{attribute addProperty BoxType "EK1100-0000-0018"}
{attribute addProperty Id "Beckhoff_EL31xxEK1122Beckhoff_EL31xxEK1122_F35612A4162A_0001_EL3101_0000_0016EL3101_EA8DF7B012816A_0002_EL3101_0000_0017EL3101_EA8DF7B012816A_0003_EL3101_0000_0018EL3101_60464DCF12816A_0004_EL3101_0000_0019EL3101_60464DCF12816A_0005_EL3102_0000_0000EL3102_B73BDD5814418A_0006_EL3102_0000_0016EL3102_8E42B51D24430.5A_0007_EL3102_0000_0017EL3102_8E42B51D24430.5A_0008_EL3102_0000_0018EL3102_8E42B51D24430.5A_0009_EL3102_0000_0019EL3102_68FCBB3024430.5A_0010_EL3102_0000_0020EL3102_1C870F0C16020A_0011_EL3104_0000_0016EL3104_55F04E9922428A_0012_EL3104_0000_0017EL3104_55F04E9922428A_0013_EL3104_0000_0018EL3104_83515A0D22428A_0014_EL3104_0000_0019EL3104_83515A0D22428A_0015_EL3104_0000_0020EL3104_83515A0D22428A_0016_EL3111_0000_0016EL3111_EA8DF7B012816A_0017_EL3111_0000_0017EL3111_EA8DF7B012816A_0018_EL3111_0000_0018EL3111_60464DCF12816A_0019_EL3111_0000_0019EL3111_60464DCF12816A_0020_EL3111_0000_0020EL3111_60464DCF12816A_0021_EL3112_0000_0000EL3112_B73BDD5814418A_0022_EL3112_0000_0016EL3112_8E42B51D24430.5A_0023_EL3112_0000_0017EL3112_8E42B51D24430.5A_0024_EL3112_0000_0018EL3112_8E42B51D24430.5A_0025_EL3112_0000_0019EL3112_1C870F0C16020A_0026_EL3112_0011_0016EL3112_1C870F0C16020A_0027_EL3114_0000_0016EL3114_129272B139249A_0028_EL3114_0000_0017EL3114_55F04E9922428A_0029_EL3114_0000_0018EL3114_55F04E9922428A_0030_EL3114_0000_0019EL3114_83515A0D22428A_0031_EL3114_0000_0020EL3114_83515A0D22428A_0032_EL3114_0000_0021EL3114_83515A0D22428A_0033_EL3121_0000_0016EL3121_EA8DF7B012816A_0034_EL3121_0000_0017EL3121_EA8DF7B012816A_0035_EL3121_0000_0018EL3121_60464DCF12816A_0036_EL3121_0000_0019EL3121_60464DCF12816A_0037_EL3122_0000_0000EL3122_B73BDD5814418A_0038_EL3122_0000_0016EL3122_8E42B51D24430.5A_0039_EL3122_0000_0017EL3122_8E42B51D24430.5A_0040_EL3122_0000_0018EL3122_8E42B51D24430.5A_0041_EL3122_0000_0019EL3122_1C870F0C16020A_0042_EL3124_0000_0016EL3124_55F04E9922428A_0043_EL3124_0000_0017EL3124_55F04E9922428A_0044_EL3124_0000_0018EL3124_83515A0D22428A_0045_EL3124_0000_0019EL3124_83515A0D22428A_0046_EL3124_0000_0020EL3124_83515A0D22428A_0047_EL3124_0090_0016EL3124_83515A0D22428A_0048_EL3141_0000_0016EL3141_EA8DF7B012816A_0049_EL3141_0000_0017EL3141_EA8DF7B012816A_0050_EL3141_0000_0018EL3141_60464DCF12816A_0051_EL3141_0000_0019EL3141_60464DCF12816A_0052_EL3141_0000_0020EL3141_60464DCF12816A_0053_EL3142_0000_0000EL3142_B73BDD5814418A_0054_EL3142_0000_0016EL3142_8E42B51D24430.5A_0055_EL3142_0000_0017EL3142_8E42B51D24430.5A_0056_EL3142_0000_0018EL3142_8E42B51D24430.5A_0057_EL3142_0000_0019EL3142_1C870F0C16020A_0058_EL3142_0010_0000EL3142_B73BDD5814418A_0059_EL3142_0010_0016EL3142_8E42B51D24430.5A_0060_EL3142_0010_0017EL3142_8E42B51D24430.5A_0061_EL3142_0010_0018EL3142_8E42B51D24430.5A_0062_EL3142_0010_0019EL3142_8E42B51D24430.5A_0063_EL3142_0010_0020EL3142_1C870F0C16020A_0064_EL3142_0010_0021EL3142_1C870F0C16020A_0065_EL3144_0000_0016EL3144_55F04E9922428A_0066_EL3144_0000_0017EL3144_55F04E9922428A_0067_EL3144_0000_0018EL3144_83515A0D22428A_0068_EL3144_0000_0019EL3144_83515A0D22428A_0069_EL3144_0000_0020EL3144_83515A0D22428A_0070_EL3151_0000_0016EL3151_50D9316A17021.25A_0071_EL3151_0000_0017EL3151_50D9316A17021.25A_0072_EL3151_0000_0018EL3151_60464DCF12816A_0073_EL3151_0000_0019EL3151_60464DCF12816A_0074_EL3151_0000_0020EL3151_60464DCF12816A_0075_EL3152_0000_0000EL3152_B73BDD5814418A_0076_EL3152_0000_0016EL3152_8E42B51D24430.5A_0077_EL3152_0000_0017EL3152_8E42B51D24430.5A_0078_EL3152_0000_0018EL3152_8E42B51D24430.5A_0079_EL3152_0000_0019EL3152_1C870F0C16020A_0080_EL3154_0000_0016EL3154_55F04E9922428A_0081_EL3154_0000_0017EL3154_55F04E9922428A_0082_EL3154_0000_0018EL3154_83515A0D22428A_0083_EL3154_0000_0019EL3154_83515A0D22428A_0084_EL3154_0000_0020EL3154_83515A0D22428A_0085_EL3161_0000_0016EL3161_EA8DF7B012816A_0086_EL3161_0000_0017EL3161_EA8DF7B012816A_0087_EL3161_0000_0018EL3161_60464DCF12816A_0088_EL3161_0000_0019EL3161_60464DCF12816A_0089_EL3162_0000_0000EL3162_B73BDD5814418A_0090_EL3162_0000_0016EL3162_8E42B51D24430.5A_0091_EL3162_0000_0017EL3162_8E42B51D24430.5A_0092_EL3162_0000_0018EL3162_8E42B51D24430.5A_0093_EL3162_0000_0019EL3162_1C870F0C16020A_0094_EL3164_0000_0016EL3164_55F04E9922428A_0095_EL3164_0000_0017EL3164_55F04E9922428A_0096_EL3164_0000_0018EL3164_83515A0D22428A_0097_EL3164_0000_0019EL3164_83515A0D22428A_0098_EL3164_0000_0020EL3164_83515A0D22428A_0099_EL3174_0000_0016EL3174_83515A0D22428A_0100_EL3174_0002_0017EL3174_83515A0D22428A_0101_EL3174_0032_0016EL3174_83515A0D22428A_0102_EL3174_0090_0016EL3174_83515A0D22428A_0103_EL3182_0000_0016EL3182_8DBFD1BF20826A_0104_EL3182_0000_0017EL3182_8DBFD1BF20826"}
{attribute addProperty CRC "413625809"}
{attribute addProperty SizeInBites "20264"}
{attribute addProperty SizeInBytes "2533"}
TYPE Beckhoff_EL31xx_18A76DD1 EXTENDS EK1100_179A0949 :
STRUCT
	{attribute addProperty Name "Beckhoff_EL31xxEK1122"}
	Beckhoff_EL31xxEK1122 : Beckhoff_EL31xxEK1122_F35612A4;
	{attribute addProperty Name "A_0001_EL3101_0000_0016"}
	A_0001_EL3101_0000_0016 : EL3101_EA8DF7B0;
	{attribute addProperty Name "A_0002_EL3101_0000_0017"}
	A_0002_EL3101_0000_0017 : EL3101_EA8DF7B0;
	{attribute addProperty Name "A_0003_EL3101_0000_0018"}
	A_0003_EL3101_0000_0018 : EL3101_60464DCF;
	{attribute addProperty Name "A_0004_EL3101_0000_0019"}
	A_0004_EL3101_0000_0019 : EL3101_60464DCF;
	{attribute addProperty Name "A_0005_EL3102_0000_0000"}
	A_0005_EL3102_0000_0000 : EL3102_B73BDD58;
	{attribute addProperty Name "A_0006_EL3102_0000_0016"}
	A_0006_EL3102_0000_0016 : EL3102_8E42B51D;
	{attribute addProperty Name "A_0007_EL3102_0000_0017"}
	A_0007_EL3102_0000_0017 : EL3102_8E42B51D;
	{attribute addProperty Name "A_0008_EL3102_0000_0018"}
	A_0008_EL3102_0000_0018 : EL3102_8E42B51D;
	{attribute addProperty Name "A_0009_EL3102_0000_0019"}
	A_0009_EL3102_0000_0019 : EL3102_68FCBB30;
	{attribute addProperty Name "A_0010_EL3102_0000_0020"}
	A_0010_EL3102_0000_0020 : EL3102_1C870F0C;
	{attribute addProperty Name "A_0011_EL3104_0000_0016"}
	A_0011_EL3104_0000_0016 : EL3104_55F04E99;
	{attribute addProperty Name "A_0012_EL3104_0000_0017"}
	A_0012_EL3104_0000_0017 : EL3104_55F04E99;
	{attribute addProperty Name "A_0013_EL3104_0000_0018"}
	A_0013_EL3104_0000_0018 : EL3104_83515A0D;
	{attribute addProperty Name "A_0014_EL3104_0000_0019"}
	A_0014_EL3104_0000_0019 : EL3104_83515A0D;
	{attribute addProperty Name "A_0015_EL3104_0000_0020"}
	A_0015_EL3104_0000_0020 : EL3104_83515A0D;
	{attribute addProperty Name "A_0016_EL3111_0000_0016"}
	A_0016_EL3111_0000_0016 : EL3111_EA8DF7B0;
	{attribute addProperty Name "A_0017_EL3111_0000_0017"}
	A_0017_EL3111_0000_0017 : EL3111_EA8DF7B0;
	{attribute addProperty Name "A_0018_EL3111_0000_0018"}
	A_0018_EL3111_0000_0018 : EL3111_60464DCF;
	{attribute addProperty Name "A_0019_EL3111_0000_0019"}
	A_0019_EL3111_0000_0019 : EL3111_60464DCF;
	{attribute addProperty Name "A_0020_EL3111_0000_0020"}
	A_0020_EL3111_0000_0020 : EL3111_60464DCF;
	{attribute addProperty Name "A_0021_EL3112_0000_0000"}
	A_0021_EL3112_0000_0000 : EL3112_B73BDD58;
	{attribute addProperty Name "A_0022_EL3112_0000_0016"}
	A_0022_EL3112_0000_0016 : EL3112_8E42B51D;
	{attribute addProperty Name "A_0023_EL3112_0000_0017"}
	A_0023_EL3112_0000_0017 : EL3112_8E42B51D;
	{attribute addProperty Name "A_0024_EL3112_0000_0018"}
	A_0024_EL3112_0000_0018 : EL3112_8E42B51D;
	{attribute addProperty Name "A_0025_EL3112_0000_0019"}
	A_0025_EL3112_0000_0019 : EL3112_1C870F0C;
	{attribute addProperty Name "A_0026_EL3112_0011_0016"}
	A_0026_EL3112_0011_0016 : EL3112_1C870F0C;
	{attribute addProperty Name "A_0027_EL3114_0000_0016"}
	A_0027_EL3114_0000_0016 : EL3114_129272B1;
	{attribute addProperty Name "A_0028_EL3114_0000_0017"}
	A_0028_EL3114_0000_0017 : EL3114_55F04E99;
	{attribute addProperty Name "A_0029_EL3114_0000_0018"}
	A_0029_EL3114_0000_0018 : EL3114_55F04E99;
	{attribute addProperty Name "A_0030_EL3114_0000_0019"}
	A_0030_EL3114_0000_0019 : EL3114_83515A0D;
	{attribute addProperty Name "A_0031_EL3114_0000_0020"}
	A_0031_EL3114_0000_0020 : EL3114_83515A0D;
	{attribute addProperty Name "A_0032_EL3114_0000_0021"}
	A_0032_EL3114_0000_0021 : EL3114_83515A0D;
	{attribute addProperty Name "A_0033_EL3121_0000_0016"}
	A_0033_EL3121_0000_0016 : EL3121_EA8DF7B0;
	{attribute addProperty Name "A_0034_EL3121_0000_0017"}
	A_0034_EL3121_0000_0017 : EL3121_EA8DF7B0;
	{attribute addProperty Name "A_0035_EL3121_0000_0018"}
	A_0035_EL3121_0000_0018 : EL3121_60464DCF;
	{attribute addProperty Name "A_0036_EL3121_0000_0019"}
	A_0036_EL3121_0000_0019 : EL3121_60464DCF;
	{attribute addProperty Name "A_0037_EL3122_0000_0000"}
	A_0037_EL3122_0000_0000 : EL3122_B73BDD58;
	{attribute addProperty Name "A_0038_EL3122_0000_0016"}
	A_0038_EL3122_0000_0016 : EL3122_8E42B51D;
	{attribute addProperty Name "A_0039_EL3122_0000_0017"}
	A_0039_EL3122_0000_0017 : EL3122_8E42B51D;
	{attribute addProperty Name "A_0040_EL3122_0000_0018"}
	A_0040_EL3122_0000_0018 : EL3122_8E42B51D;
	{attribute addProperty Name "A_0041_EL3122_0000_0019"}
	A_0041_EL3122_0000_0019 : EL3122_1C870F0C;
	{attribute addProperty Name "A_0042_EL3124_0000_0016"}
	A_0042_EL3124_0000_0016 : EL3124_55F04E99;
	{attribute addProperty Name "A_0043_EL3124_0000_0017"}
	A_0043_EL3124_0000_0017 : EL3124_55F04E99;
	{attribute addProperty Name "A_0044_EL3124_0000_0018"}
	A_0044_EL3124_0000_0018 : EL3124_83515A0D;
	{attribute addProperty Name "A_0045_EL3124_0000_0019"}
	A_0045_EL3124_0000_0019 : EL3124_83515A0D;
	{attribute addProperty Name "A_0046_EL3124_0000_0020"}
	A_0046_EL3124_0000_0020 : EL3124_83515A0D;
	{attribute addProperty Name "A_0047_EL3124_0090_0016"}
	A_0047_EL3124_0090_0016 : EL3124_83515A0D;
	{attribute addProperty Name "A_0048_EL3141_0000_0016"}
	A_0048_EL3141_0000_0016 : EL3141_EA8DF7B0;
	{attribute addProperty Name "A_0049_EL3141_0000_0017"}
	A_0049_EL3141_0000_0017 : EL3141_EA8DF7B0;
	{attribute addProperty Name "A_0050_EL3141_0000_0018"}
	A_0050_EL3141_0000_0018 : EL3141_60464DCF;
	{attribute addProperty Name "A_0051_EL3141_0000_0019"}
	A_0051_EL3141_0000_0019 : EL3141_60464DCF;
	{attribute addProperty Name "A_0052_EL3141_0000_0020"}
	A_0052_EL3141_0000_0020 : EL3141_60464DCF;
	{attribute addProperty Name "A_0053_EL3142_0000_0000"}
	A_0053_EL3142_0000_0000 : EL3142_B73BDD58;
	{attribute addProperty Name "A_0054_EL3142_0000_0016"}
	A_0054_EL3142_0000_0016 : EL3142_8E42B51D;
	{attribute addProperty Name "A_0055_EL3142_0000_0017"}
	A_0055_EL3142_0000_0017 : EL3142_8E42B51D;
	{attribute addProperty Name "A_0056_EL3142_0000_0018"}
	A_0056_EL3142_0000_0018 : EL3142_8E42B51D;
	{attribute addProperty Name "A_0057_EL3142_0000_0019"}
	A_0057_EL3142_0000_0019 : EL3142_1C870F0C;
	{attribute addProperty Name "A_0058_EL3142_0010_0000"}
	A_0058_EL3142_0010_0000 : EL3142_B73BDD58;
	{attribute addProperty Name "A_0059_EL3142_0010_0016"}
	A_0059_EL3142_0010_0016 : EL3142_8E42B51D;
	{attribute addProperty Name "A_0060_EL3142_0010_0017"}
	A_0060_EL3142_0010_0017 : EL3142_8E42B51D;
	{attribute addProperty Name "A_0061_EL3142_0010_0018"}
	A_0061_EL3142_0010_0018 : EL3142_8E42B51D;
	{attribute addProperty Name "A_0062_EL3142_0010_0019"}
	A_0062_EL3142_0010_0019 : EL3142_8E42B51D;
	{attribute addProperty Name "A_0063_EL3142_0010_0020"}
	A_0063_EL3142_0010_0020 : EL3142_1C870F0C;
	{attribute addProperty Name "A_0064_EL3142_0010_0021"}
	A_0064_EL3142_0010_0021 : EL3142_1C870F0C;
	{attribute addProperty Name "A_0065_EL3144_0000_0016"}
	A_0065_EL3144_0000_0016 : EL3144_55F04E99;
	{attribute addProperty Name "A_0066_EL3144_0000_0017"}
	A_0066_EL3144_0000_0017 : EL3144_55F04E99;
	{attribute addProperty Name "A_0067_EL3144_0000_0018"}
	A_0067_EL3144_0000_0018 : EL3144_83515A0D;
	{attribute addProperty Name "A_0068_EL3144_0000_0019"}
	A_0068_EL3144_0000_0019 : EL3144_83515A0D;
	{attribute addProperty Name "A_0069_EL3144_0000_0020"}
	A_0069_EL3144_0000_0020 : EL3144_83515A0D;
	{attribute addProperty Name "A_0070_EL3151_0000_0016"}
	A_0070_EL3151_0000_0016 : EL3151_50D9316A;
	{attribute addProperty Name "A_0071_EL3151_0000_0017"}
	A_0071_EL3151_0000_0017 : EL3151_50D9316A;
	{attribute addProperty Name "A_0072_EL3151_0000_0018"}
	A_0072_EL3151_0000_0018 : EL3151_60464DCF;
	{attribute addProperty Name "A_0073_EL3151_0000_0019"}
	A_0073_EL3151_0000_0019 : EL3151_60464DCF;
	{attribute addProperty Name "A_0074_EL3151_0000_0020"}
	A_0074_EL3151_0000_0020 : EL3151_60464DCF;
	{attribute addProperty Name "A_0075_EL3152_0000_0000"}
	A_0075_EL3152_0000_0000 : EL3152_B73BDD58;
	{attribute addProperty Name "A_0076_EL3152_0000_0016"}
	A_0076_EL3152_0000_0016 : EL3152_8E42B51D;
	{attribute addProperty Name "A_0077_EL3152_0000_0017"}
	A_0077_EL3152_0000_0017 : EL3152_8E42B51D;
	{attribute addProperty Name "A_0078_EL3152_0000_0018"}
	A_0078_EL3152_0000_0018 : EL3152_8E42B51D;
	{attribute addProperty Name "A_0079_EL3152_0000_0019"}
	A_0079_EL3152_0000_0019 : EL3152_1C870F0C;
	{attribute addProperty Name "A_0080_EL3154_0000_0016"}
	A_0080_EL3154_0000_0016 : EL3154_55F04E99;
	{attribute addProperty Name "A_0081_EL3154_0000_0017"}
	A_0081_EL3154_0000_0017 : EL3154_55F04E99;
	{attribute addProperty Name "A_0082_EL3154_0000_0018"}
	A_0082_EL3154_0000_0018 : EL3154_83515A0D;
	{attribute addProperty Name "A_0083_EL3154_0000_0019"}
	A_0083_EL3154_0000_0019 : EL3154_83515A0D;
	{attribute addProperty Name "A_0084_EL3154_0000_0020"}
	A_0084_EL3154_0000_0020 : EL3154_83515A0D;
	{attribute addProperty Name "A_0085_EL3161_0000_0016"}
	A_0085_EL3161_0000_0016 : EL3161_EA8DF7B0;
	{attribute addProperty Name "A_0086_EL3161_0000_0017"}
	A_0086_EL3161_0000_0017 : EL3161_EA8DF7B0;
	{attribute addProperty Name "A_0087_EL3161_0000_0018"}
	A_0087_EL3161_0000_0018 : EL3161_60464DCF;
	{attribute addProperty Name "A_0088_EL3161_0000_0019"}
	A_0088_EL3161_0000_0019 : EL3161_60464DCF;
	{attribute addProperty Name "A_0089_EL3162_0000_0000"}
	A_0089_EL3162_0000_0000 : EL3162_B73BDD58;
	{attribute addProperty Name "A_0090_EL3162_0000_0016"}
	A_0090_EL3162_0000_0016 : EL3162_8E42B51D;
	{attribute addProperty Name "A_0091_EL3162_0000_0017"}
	A_0091_EL3162_0000_0017 : EL3162_8E42B51D;
	{attribute addProperty Name "A_0092_EL3162_0000_0018"}
	A_0092_EL3162_0000_0018 : EL3162_8E42B51D;
	{attribute addProperty Name "A_0093_EL3162_0000_0019"}
	A_0093_EL3162_0000_0019 : EL3162_1C870F0C;
	{attribute addProperty Name "A_0094_EL3164_0000_0016"}
	A_0094_EL3164_0000_0016 : EL3164_55F04E99;
	{attribute addProperty Name "A_0095_EL3164_0000_0017"}
	A_0095_EL3164_0000_0017 : EL3164_55F04E99;
	{attribute addProperty Name "A_0096_EL3164_0000_0018"}
	A_0096_EL3164_0000_0018 : EL3164_83515A0D;
	{attribute addProperty Name "A_0097_EL3164_0000_0019"}
	A_0097_EL3164_0000_0019 : EL3164_83515A0D;
	{attribute addProperty Name "A_0098_EL3164_0000_0020"}
	A_0098_EL3164_0000_0020 : EL3164_83515A0D;
	{attribute addProperty Name "A_0099_EL3174_0000_0016"}
	A_0099_EL3174_0000_0016 : EL3174_83515A0D;
	{attribute addProperty Name "A_0100_EL3174_0002_0017"}
	A_0100_EL3174_0002_0017 : EL3174_83515A0D;
	{attribute addProperty Name "A_0101_EL3174_0032_0016"}
	A_0101_EL3174_0032_0016 : EL3174_83515A0D;
	{attribute addProperty Name "A_0102_EL3174_0090_0016"}
	A_0102_EL3174_0090_0016 : EL3174_83515A0D;
	{attribute addProperty Name "A_0103_EL3182_0000_0016"}
	A_0103_EL3182_0000_0016 : EL3182_8DBFD1BF;
	{attribute addProperty Name "A_0104_EL3182_0000_0017"}
	A_0104_EL3182_0000_0017 : EL3182_8DBFD1BF;
END_STRUCT
END_TYPE

(* stored: Version 1.2.0.0, ProductVersion 3.1.4024.9
   DUT Beckhoff_EL31xx_18A76DD1: Id {96149751-fed4-4bdb-9399-5034e46ab33e} *)
